(* CODESYS project 1a.project

Project tree, tasks and I/O mapping:
  Device : CODESYS Control Win V3, 3S - Smart Software Solutions GmbH, order no. 305021, version 3.5.11.30
    application Application
      libraries: Standard, * (System)
      task MainTask (cyclic, interval t#20ms, priority 1) calls PLC_PRG
      program PLC_PRG [LD]
*)

// Device/Application/PLC_PRG
PROGRAM PLC_PRG
VAR 
	b1: BOOL;
	b2: BOOL;
	k1: BOOL;
	k2: BOOL;
END_VAR

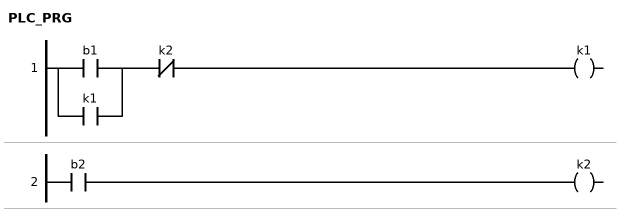
// NETWORK 1
k1 := (b1 OR k1) AND NOT k2;

// NETWORK 2
k2 := b2;

END_PROGRAM
